TEXTLIST CommandOnTerminalEvent
  0 = 'Do Nothing'
  1 = 'Off'
  2 = 'RecallMaxLevel'
  3 = 'RecallMinLevel'
  4 = 'GoToScene0'
  5 = 'GoToScene1'
  6 = 'GoToScene2'
  7 = 'GoToScene3'
  8 = 'GoToScene4'
  9 = 'GoToScene5'
  10 = 'GoToScene6'
  11 = 'GoToScene7'
  12 = 'GoToScene8'
  13 = 'GoToScene9'
  14 = 'GoToScene10'
  15 = 'GoToScene11'
  16 = 'GoToScene12'
  17 = 'GoToScene13'
  18 = 'GoToScene14'
  19 = 'GoToScene15'
   = ''
END_TEXTLIST

(* stored: Version 1.1.0.1, ProductVersion 3.1.4024.4
   TextList CommandOnTerminalEvent: Id {1816ff85-34a2-4552-bf1a-2bb771aeb34c} *)
